SUBAPPLICATION Uebung_011b7_AX (* Numeric Value Input SAFE_DIV *)
  (* Standard: 61499-2; Description: Copyright (c) 2026 Meisterschulen am Ostbahnhof This program and the accompanying materials are made available under the terms of the Eclipse Public License 2.0 which is available at https://www.eclipse.org/legal/epl-2.0/ SPDX-License-Identifier: EPL-2.0 *)
  (* Version 1.0, 2026-09-10, Franz Höpfinger, Meisterschulen am Ostbahnhof, initial API and implementation and/or initial documentation *)
  PACKAGE Uebungen;
  IMPORT Uebungen::const::UT::DefaultPool::InputNumber_I1;
  IMPORT Uebungen::const::UT::DefaultPool::InputNumber_I2;
  IMPORT Uebungen::const::UT::DefaultPool::OutputNumber_N1;
  IMPORT Uebungen::const::UT::DefaultPool::OutputNumber_N2;
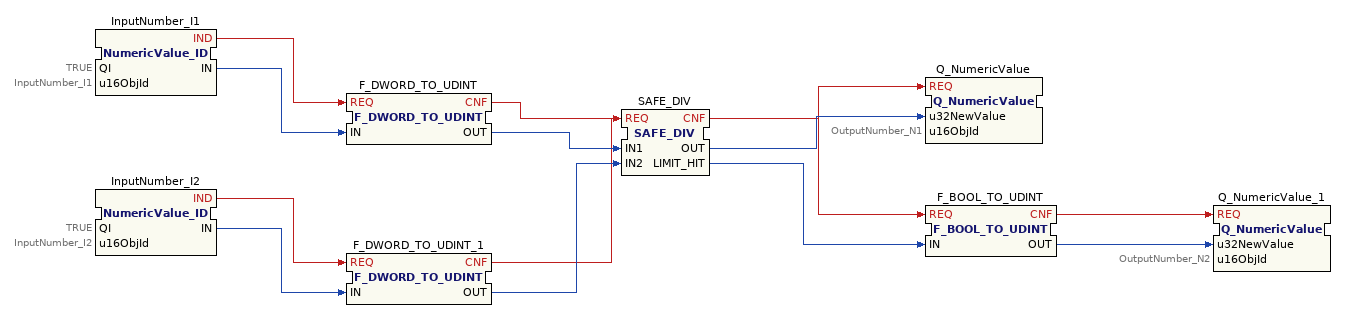
  FBS
    InputNumber_I1 : isobus::UT::io::NumericValue::NumericValue_ID(QI := TRUE, u16ObjId := InputNumber_I1);
    InputNumber_I2 : isobus::UT::io::NumericValue::NumericValue_ID(QI := TRUE, u16ObjId := InputNumber_I2);
    F_DWORD_TO_UDINT : iec61131::conversion::F_DWORD_TO_UDINT;
    F_DWORD_TO_UDINT_1 : iec61131::conversion::F_DWORD_TO_UDINT;
    SAFE_DIV : SafeArithmetic::arithmetic::SAFE_DIV;
    Q_NumericValue : isobus::UT::Q::Q_NumericValue(u16ObjId := OutputNumber_N1);
    F_BOOL_TO_UDINT : iec61131::conversion::F_BOOL_TO_UDINT;
    Q_NumericValue_1 : isobus::UT::Q::Q_NumericValue(u16ObjId := OutputNumber_N2);
  END_FBS
  EVENT_CONNECTIONS
    InputNumber_I1.IND TO F_DWORD_TO_UDINT.REQ;
    InputNumber_I2.IND TO F_DWORD_TO_UDINT_1.REQ;
    F_DWORD_TO_UDINT.CNF TO SAFE_DIV.REQ;
    F_DWORD_TO_UDINT_1.CNF TO SAFE_DIV.REQ;
    SAFE_DIV.CNF TO Q_NumericValue.REQ;
    SAFE_DIV.CNF TO F_BOOL_TO_UDINT.REQ;
    F_BOOL_TO_UDINT.CNF TO Q_NumericValue_1.REQ;
  END_CONNECTIONS
  DATA_CONNECTIONS
    InputNumber_I1.IN TO F_DWORD_TO_UDINT.IN;
    InputNumber_I2.IN TO F_DWORD_TO_UDINT_1.IN;
    F_DWORD_TO_UDINT.OUT TO SAFE_DIV.IN1;
    F_DWORD_TO_UDINT_1.OUT TO SAFE_DIV.IN2;
    SAFE_DIV.OUT TO Q_NumericValue.u32NewValue;
    SAFE_DIV.LIMIT_HIT TO F_BOOL_TO_UDINT.IN;
    F_BOOL_TO_UDINT.OUT TO Q_NumericValue_1.u32NewValue;
  END_CONNECTIONS
END_SUBAPPLICATION
